// Composition root instance. Its members are already private (attributes in
// FB_SpkMain); whether the DB itself can also be hidden from OPC UA by a source
// attribute or only by the block property is settled in S1 (Part IV s.3.10.1).
DATA_BLOCK "SpkMain"
{ S7_Optimized_Access := 'TRUE' }
VERSION : 0.1
NON_RETAIN
"FB_SpkMain"

BEGIN

END_DATA_BLOCK
